FUNCTION_BLOCK FT_DERIV_AR (* AR-Adapter-Wrapper um OSCAT FT_DERIV - bruckt zwischen adapter und OSCAT, ohne dass eine der beiden Basisbibliotheken von der anderen abhaengt. K/run als Klartext-InputVars durchgereicht (Default K=1.0, run=TRUE) *)
  (* Standard: 61499-2; Description: Copyright (c) 2026 Meisterschulen am Ostbahnhof This program and the accompanying materials are made available under the terms of the Eclipse Public License 2.0 which is available at https://www.eclipse.org/legal/epl-2.0/ SPDX-License-Identifier: EPL-2.0 *)
  (* Version 1.4, 2026-09-20, Franz Höpfinger, Meisterschulen am Ostbahnhof, Bugfix: K/run wurden nur per plain DataConnection an FT_DERIV durchgereicht, ausgeloest einzig ueber AR_IN.E1 - kein Event auf diesem Wrapper hatte je eine With-Verknuepfung fuer diese Vars (IEC 61499 - ungebundene Vars werden nicht zuverlaessig gelesen). Neues explizites REQ-EventInput ergaenzt (parallel zu AR_IN.E1, beide -> FT_DERIV.REQ) mit With K/run. *)
  (* Version 1.3, 2026-08-30, Franz Höpfinger, Meisterschulen am Ostbahnhof, Reine Adapter-Grenze: delta_t/delta_in als eigene Adapter (AUDI/AR) statt Klartext-Event; K/run als Klartext-InputVars durchgereicht, kein Adapter noetig, da beides pro Aufruf konstant ist *)
  PACKAGE OSCAT_adapter::Control;
  (* Documentation:
  FT_DERIV_AR
   🇩🇪 Deutsch
   AR-Adapter-Wrapper um OSCAT::Basic::POUs::Engineering::Control::FT_DERIV. K (Ableitungsfaktor, Default 1.0) und run (Berechnung aktiv, Default TRUE) sind Klartext-InputVars auf diesem Wrapper. Ein explizites REQ-EventInput (mit With K und With run) erlaubt den manuellen/periodischen Aufruf zusaetzlich zum automatischen Ausloesen ueber AR_IN.E1 (IEC 61499 - With-Verknuepfung fuer zuverlaessiges Einlesen der Parameter).
   Reine Adapter-Grenze
   Alle drei von FT_DERIV gelieferten Werte werden als eigene Adapter exponiert - kein Klartext-Event/-Datum verlaesst diesen Baustein:
    - AR_OUT (Plug, AR): die berechnete Ableitung (out, REAL)
   - AR_DELTA_IN (Plug, AR): Differenz des Eingangssignals (delta_in, REAL)
   - AUDI_DELTA_T (Plug, AUDI): Zeitdifferenz in Mikrosekunden (delta_t, UDINT - AUDI ist der passende Adapter-Typ fuer UDINT)
    INIT/INITO und RST werden 1:1 an FT_DERIV.EINIT/.INITO/.RST durchgereicht - wie bei den uebrigen Service-Wrappern in diesem Repo (z. B. Q_NumericValue_AUDI, logiBUS_PI_IDA), damit Lebenszyklus und Reset auch fuer diesen Baustein von aussen ansteuerbar sind. Bleibt INIT unverdrahtet, feuert es einmalig beim Deployment automatisch (Standardkonvention fuer unverdrahtete EInit-Events).
   Braucht eine aufrufende Komposition einen Klartext-Wert (z. B. fuer Q_NumericValue_PHYS.rPhys, das keinen Adapter hat), wird dafuer der bereits vorhandene generische Baustein adapter::conversion::unidirectional::AR_R_TO_REAL verwendet (Socket AR_IN -> Klartext-CNF/IN) - nicht ein eigener Klartext-Ausgang an diesem Wrapper.
   Warum ein eigener Wrapper (und nicht direkt FT_DERIV in der Komposition verdrahten)?
   FT_DERIV ist ein reines OSCAT-FB ohne Adapter-Schnittstelle (REQ/CNF sind einfache Events, keine AR-Sockets/Plugs). Ein einzelnes Roh-Sub-Signal (.E1/.D1) eines FREMD-instanzierten Adapter-Bausteins (z. B. AD_TO_AR_NUM.AR_OUT) laesst sich in einem uebergeordneten SubApp-Netzwerk NICHT direkt an ein einfaches Event/Datum eines anderen, ebenfalls fremd-instanzierten FBs verdrahten - diese .E1/.D1-Zugriffssyntax ist nur INNERHALB der Definition eines FBTyps fuer dessen EIGENE Grenz-Sockets/-Plugs gueltig (siehe z. B. Q_NumericValue_AUDI, das genau so intern Q_NumericValue einwickelt).
   Zugleich soll adapter nicht von OSCAT abhaengen (und umgekehrt) - beide sollen unabhaengige, generische Basisbibliotheken bleiben. Die Loesung: ein DRITTES, eigenes Bibliotheks-Projekt (OSCAT_adapter), das von BEIDEN abhaengt und die Bruecke in einem eigenen FBTyp kapselt - mit einer rein adapter-basierten Aussengrenze, damit auch dieser Baustein selbst wieder ganz normal ueber AdapterConnections mit anderen AR/AUDI-Bausteinen verbunden werden kann (kein .E1/.D1 noetig).
   🇬🇧 English
   AR-adapter wrapper around OSCAT::Basic::POUs::Engineering::Control::FT_DERIV. K (derivation factor, default 1.0) and run (calculation enabled, default TRUE) are plain InputVars on this wrapper. An explicit REQ event input (with With K and With run bindings) enables manual or periodic execution in addition to automatic triggering via AR_IN.E1 (per IEC 61499, binding input variables via With for reliable reading).
   Pure adapter boundary
   All three values FT_DERIV produces are exposed as their own adapters - no plain event/data leaves this block:
    - AR_OUT (plug, AR): the calculated derivative (out, REAL)
   - AR_DELTA_IN (plug, AR): input signal difference (delta_in, REAL)
   - AUDI_DELTA_T (plug, AUDI): time difference in microseconds (delta_t, UDINT - AUDI is the matching adapter type for UDINT)
    INIT/INITO and RST are passed through 1:1 to FT_DERIV.EINIT/.INITO/.RST - as with the other service wrappers in this repo (e.g. Q_NumericValue_AUDI, logiBUS_PI_IDA), so lifecycle and reset remain controllable from the outside. If INIT is left unconnected, it auto-fires once at deployment (standard convention for unconnected EInit events).
   If a calling composition needs a plain value (e.g. for Q_NumericValue_PHYS.rPhys, which has no adapter), it uses the existing generic block adapter::conversion::unidirectional::AR_R_TO_REAL for that (socket AR_IN -> plain CNF/IN) - not a dedicated plain output on this wrapper.
   Why a dedicated wrapper (instead of wiring FT_DERIV directly into a composition)?
   FT_DERIV is a plain OSCAT FB with no adapter interface (REQ/CNF are ordinary events, not AR sockets/plugs). A raw sub-signal (.E1/.D1) of an EXTERNALLY instantiated adapter FB (e.g. AD_TO_AR_NUM.AR_OUT) cannot be wired directly, from a parent SubApp network, into a plain event/data pin of another externally instantiated FB - this .E1/.D1 access syntax is only valid INSIDE an FBType's own definition, for its OWN boundary sockets/plugs (see e.g. Q_NumericValue_AUDI, which wraps Q_NumericValue internally in exactly this way).
   At the same time, adapter must not depend on OSCAT (nor vice versa) - both should stay independent, generic base libraries. The solution: a THIRD, dedicated library project (OSCAT_adapter) that depends on BOTH and encapsulates the bridge in its own FBType, with a purely adapter-based outer boundary so this block itself can again be wired up via ordinary AdapterConnections to other AR/AUDI blocks (no .E1/.D1 needed).
  *)
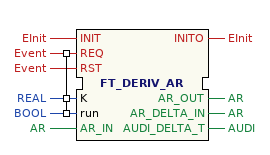
  EVENT_INPUT
    INIT : EInit; (* Service Initialization (durchgereicht an FT_DERIV.EINIT) *)
    REQ WITH K, run; (* Explizite Ausfuehrungsanforderung (durchgereicht an FT_DERIV.REQ, zusaetzlich zu AR_IN.E1) *)
    RST; (* Reset der Ableitungshistorie (durchgereicht an FT_DERIV.RST) *)
  END_EVENT
  EVENT_OUTPUT
    INITO : EInit; (* Initialization Confirm *)
  END_EVENT
  VAR_INPUT
    K : REAL := 1.0; (* Ableitungsfaktor (durchgereicht an FT_DERIV.K) *)
    run : BOOL := TRUE; (* Berechnung aktiv (durchgereicht an FT_DERIV.run) *)
  END_VAR
  SOCKETS
    AR_IN : adapter::types::unidirectional::AR; (* Eingangssignal (REAL) *)
  END_SOCKETS
  PLUGS
    AR_OUT : adapter::types::unidirectional::AR; (* Berechnete Ableitung (REAL, bei K=1.0 direkt in Hz, wenn IN Impulse/Zaehlerstand ist) *)
    AR_DELTA_IN : adapter::types::unidirectional::AR; (* Differenz des Eingangssignals (REAL, durchgereicht von FT_DERIV.delta_in) *)
    AUDI_DELTA_T : adapter::types::unidirectional::AUDI; (* Zeitdifferenz in Mikrosekunden (UDINT, durchgereicht von FT_DERIV.delta_t) *)
  END_PLUGS
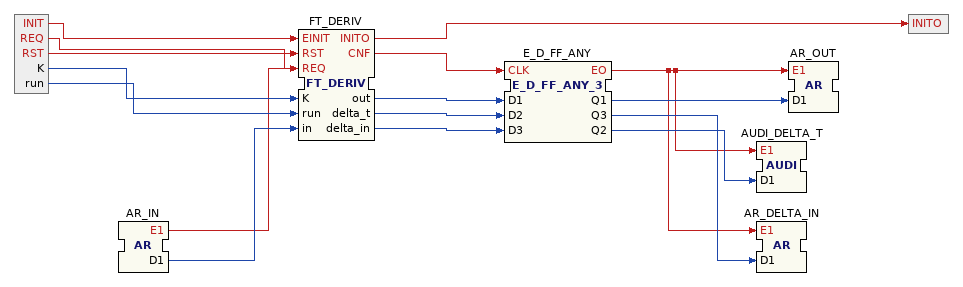
  FBS
    FT_DERIV : OSCAT::Basic::POUs::Engineering::Control::FT_DERIV;
    E_D_FF_ANY : iec61499::events::E_D_FF_ANY_3;
  END_FBS
  EVENT_CONNECTIONS
    INIT TO FT_DERIV.EINIT;
    FT_DERIV.INITO TO INITO;
    RST TO FT_DERIV.RST;
    AR_IN.E1 TO FT_DERIV.REQ;
    REQ TO FT_DERIV.REQ;
    E_D_FF_ANY.EO TO AR_OUT.E1;
    E_D_FF_ANY.EO TO AR_DELTA_IN.E1;
    E_D_FF_ANY.EO TO AUDI_DELTA_T.E1;
    FT_DERIV.CNF TO E_D_FF_ANY.CLK;
  END_CONNECTIONS
  DATA_CONNECTIONS
    K TO FT_DERIV.K;
    run TO FT_DERIV.run;
    AR_IN.D1 TO FT_DERIV.in;
    E_D_FF_ANY.Q1 TO AR_OUT.D1;
    E_D_FF_ANY.Q3 TO AR_DELTA_IN.D1;
    E_D_FF_ANY.Q2 TO AUDI_DELTA_T.D1;
    FT_DERIV.out TO E_D_FF_ANY.D1;
    FT_DERIV.delta_t TO E_D_FF_ANY.D2;
    FT_DERIV.delta_in TO E_D_FF_ANY.D3;
  END_CONNECTIONS
END_FUNCTION_BLOCK
